// TIA Portal V19 export
TYPE "MotorCtrl"
// stored: Access Published
   STRUCT
      SafeStop : Bool;   // Emergency stop (device in safe state)
      Rst : Bool;   // Reset alarms command / Reset alarms
      Run : Bool;   // Motor run request / Run command
   END_STRUCT;
END_TYPE
